(* CODESYS project sorting_by_weight.project

Project tree, tasks and I/O mapping:
  Device : CODESYS Control Win V3, 3S - Smart Software Solutions GmbH, order no. 305021, version 3.5.11.30
    application Application
      libraries: Standard, * (System)
      task MainTask (cyclic, interval t#20ms, priority 1) calls PLC_PRG
      program PLC_PRG [LD]
      Symbols
*)

// Device/Application/PLC_PRG
PROGRAM PLC_PRG
VAR
	//painel - botoes, luzes e contador
	start, stop, reset, emergency : BOOL;
	start_light, stop_light, reset_light, emergency_light: BOOL;
	
	//variaveis bool
	run, pesando : BOOL;
	leve, medio, pesado: BOOL;
	emergency_stop: BOOL;
	conveyors: BOOL;
	front: BOOL;
	left: BOOL;
	right: BOOL;
	entry_conveyor_on: BOOL;
	
	//variaveis para pesagem e contagem
	scale, weight: REAL;
	L_count, F_count, R_count : WORD;
	
	//esteiras e atuadores
	entry_conveyor, load_scale : BOOL;
	send_left, send_front, send_right: BOOL;
	left_conveyor, front_conveyor, right_conveyor : BOOL;
	
	//sensores
	at_scale_entry, at_scale, at_scale_exit: BOOL;
	at_left_entry, at_front_entry, at_right_entry : BOOL;
	at_exit_left, at_exit_front, at_exit_right : BOOL;
	
	//contadores, timers
	TON_0: TON;
	TOF_0: TOF;
	TOF_1: TOF;
	TOF_2: TOF;
	F_TRIG_0: F_TRIG;
	F_TRIG_1: F_TRIG;
	F_TRIG_2: F_TRIG;
	CTU_left: CTU;	
	CTU_front: CTU;
	CTU_right: CTU;
END_VAR
VAR // added by the converter: edge detectors and wires of the graphical bodies
    _w1, _w2, _w3, _w4, _w5, _w6 : BOOL;
    _rt1 : R_TRIG;
    _ft1 : F_TRIG;
END_VAR

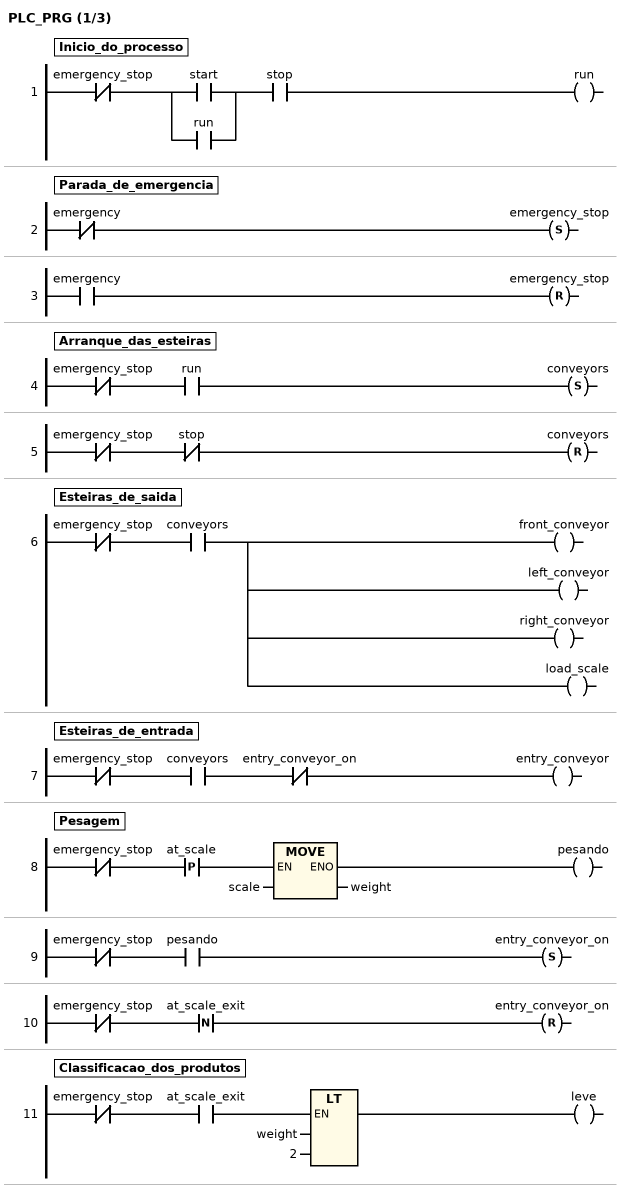
// NETWORK 1
Inicio_do_processo:
_w1 := NOT emergency_stop;
run := (_w1 AND start OR _w1 AND run) AND stop;

// NETWORK 2
Parada_de_emergencia:
emergency_stop S= NOT emergency;

// NETWORK 3
emergency_stop R= emergency;

// NETWORK 4
Arranque_das_esteiras:
conveyors S= NOT emergency_stop AND run;

// NETWORK 5
conveyors R= NOT emergency_stop AND NOT stop;

// NETWORK 6
Esteiras_de_saida:
_w2 := NOT emergency_stop AND conveyors;
front_conveyor := _w2;
left_conveyor := _w2;
right_conveyor := _w2;
load_scale := _w2;

// NETWORK 7
Esteiras_de_entrada:
entry_conveyor := NOT emergency_stop AND conveyors AND NOT entry_conveyor_on;

// NETWORK 8
Pesagem:
_rt1(CLK := at_scale);
_w3 := NOT emergency_stop AND _rt1.Q;
IF _w3 THEN weight := scale; END_IF
pesando := _w3;

// NETWORK 9
entry_conveyor_on S= NOT emergency_stop AND pesando;

// NETWORK 10
_ft1(CLK := at_scale_exit);
entry_conveyor_on R= NOT emergency_stop AND _ft1.Q;

// NETWORK 11
Classificacao_dos_produtos:
leve := NOT emergency_stop AND at_scale_exit AND weight < 2;

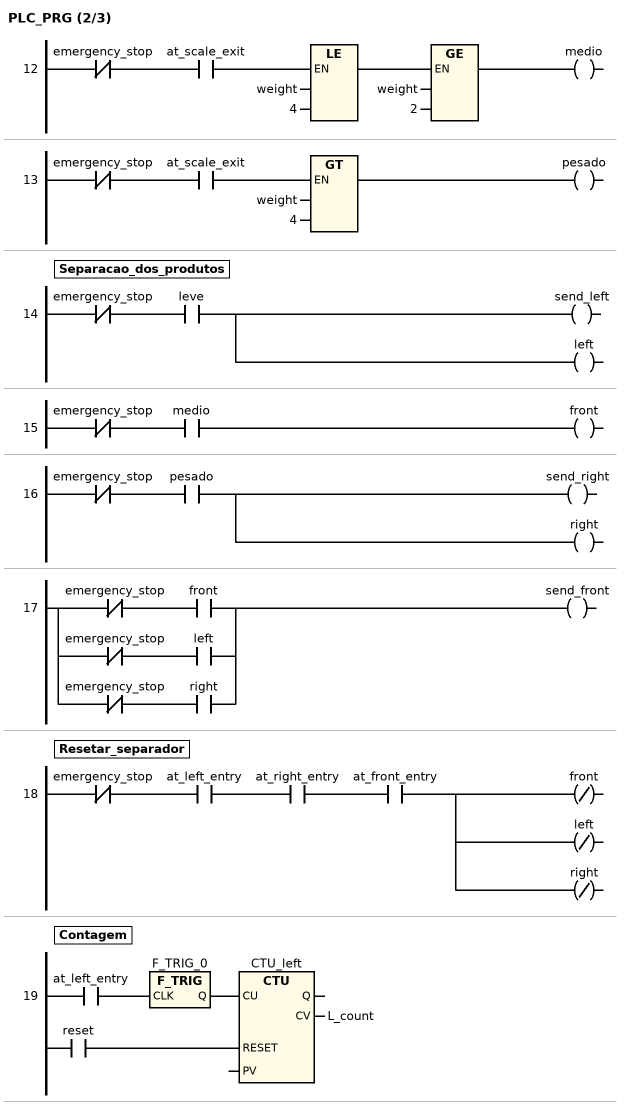
// NETWORK 12
medio := NOT emergency_stop AND at_scale_exit AND weight <= 4 AND weight >= 2;

// NETWORK 13
pesado := NOT emergency_stop AND at_scale_exit AND weight > 4;

// NETWORK 14
Separacao_dos_produtos:
_w4 := NOT emergency_stop AND leve;
send_left := _w4;
left := _w4;

// NETWORK 15
front := NOT emergency_stop AND medio;

// NETWORK 16
_w5 := NOT emergency_stop AND pesado;
send_right := _w5;
right := _w5;

// NETWORK 17
send_front := NOT emergency_stop AND front OR NOT emergency_stop AND left OR NOT emergency_stop AND right;

// NETWORK 18
Resetar_separador:
_w6 := NOT emergency_stop AND at_left_entry AND at_right_entry AND at_front_entry;
front := NOT _w6;
left := NOT _w6;
right := NOT _w6;

// NETWORK 19
Contagem:
F_TRIG_0(CLK := at_left_entry); // F_TRIG
CTU_left(CU := F_TRIG_0.Q, RESET := reset, CV => L_count); // CTU

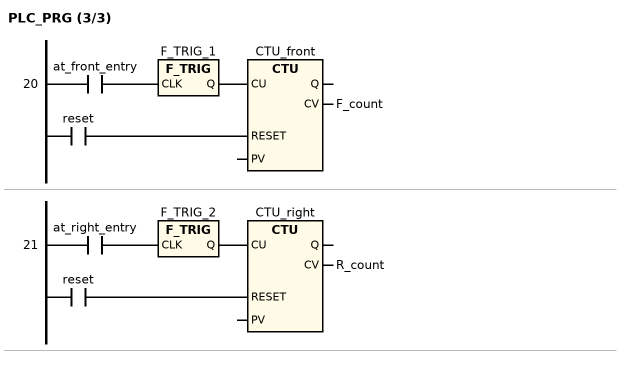
// NETWORK 20
F_TRIG_1(CLK := at_front_entry); // F_TRIG
CTU_front(CU := F_TRIG_1.Q, RESET := reset, CV => F_count); // CTU

// NETWORK 21
F_TRIG_2(CLK := at_right_entry); // F_TRIG
CTU_right(CU := F_TRIG_2.Q, RESET := reset, CV => R_count); // CTU

END_PROGRAM
